FUNCTION CheckRangeUnsigned : UDINT
VAR_INPUT
	value, lower, upper: UDINT;
END_VAR

{noflow}

IF (value < lower) THEN
	CheckRangeUnsigned := lower;
	oaksGVL.udiCheckRangeUnsigned := oaksGVL.udiCheckRangeUnsigned + 1;
ELSIF(value > upper) THEN
	CheckRangeUnsigned := upper;
	oaksGVL.udiCheckRangeUnsigned := oaksGVL.udiCheckRangeUnsigned + 1;
ELSE
	CheckRangeUnsigned := value;
END_IF
{flow}

END_FUNCTION

(* stored: Version 1.1.0.1, ProductVersion 3.1.4022.18
   POU CheckRangeUnsigned: Id {c03d91ad-ef91-4863-8bbf-b533cc79d519}, SpecialFunc CheckRangeUnsigned *)
